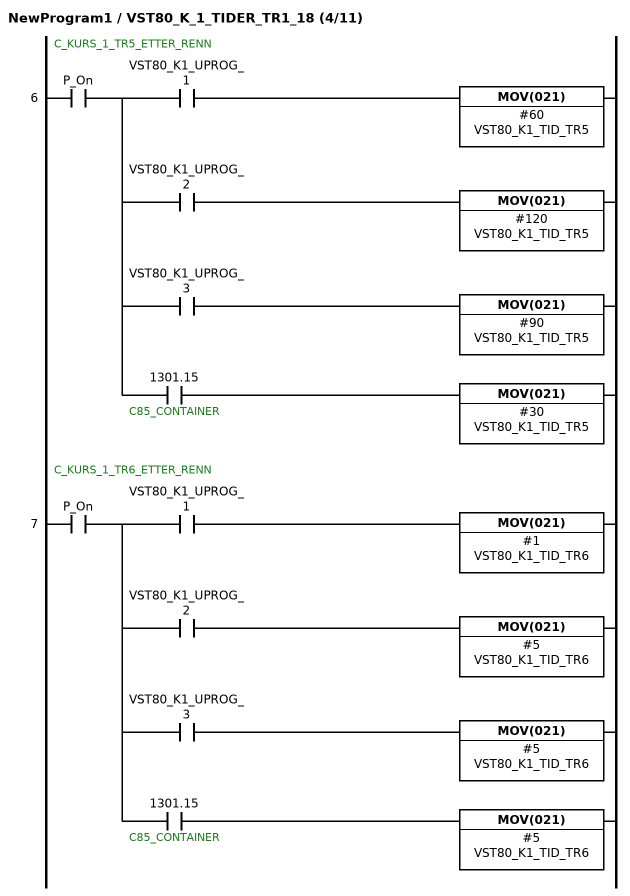
; [picture p72: NewProgram1 / VST80_K_1_TIDER_TR1_18, rungs 6-7]
; rung 6: C_KURS_1_TR5_ETTER_RENN
LD P_On
OUT TR0
AND VST80_K1_UPROG_1
MOV(021) #60 VST80_K1_TID_TR5
LD TR0
AND VST80_K1_UPROG_2
MOV(021) #120 VST80_K1_TID_TR5
LD TR0
AND VST80_K1_UPROG_3
MOV(021) #90 VST80_K1_TID_TR5
LD TR0
AND 1301.15  ; C85_CONTAINER
MOV(021) #30 VST80_K1_TID_TR5
; rung 7: C_KURS_1_TR6_ETTER_RENN
LD P_On
OUT TR0
AND VST80_K1_UPROG_1
MOV(021) #1 VST80_K1_TID_TR6
LD TR0
AND VST80_K1_UPROG_2
MOV(021) #5 VST80_K1_TID_TR6
LD TR0
AND VST80_K1_UPROG_3
MOV(021) #5 VST80_K1_TID_TR6
LD TR0
AND 1301.15  ; C85_CONTAINER
MOV(021) #5 VST80_K1_TID_TR6

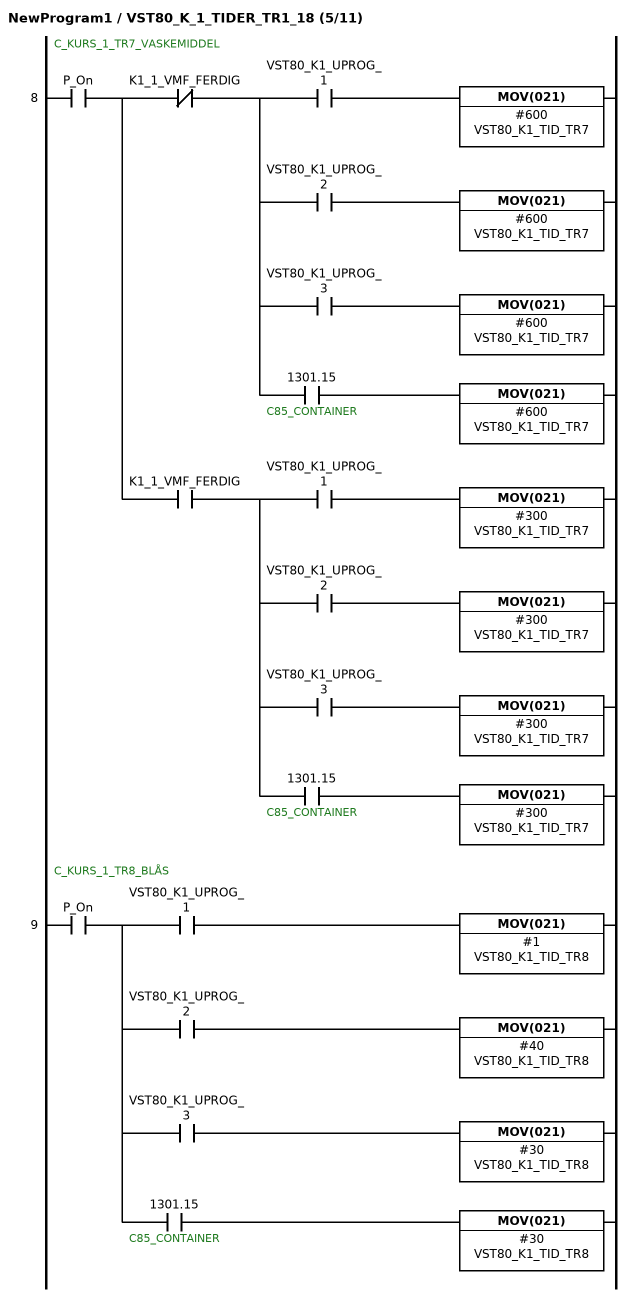
; rung 8: C_KURS_1_TR7_VASKEMIDDEL
LD P_On
OUT TR0
ANDNOT K1_1_VMF_FERDIG
OUT TR1
AND VST80_K1_UPROG_1
MOV(021) #600 VST80_K1_TID_TR7
LD TR1
AND VST80_K1_UPROG_2
MOV(021) #600 VST80_K1_TID_TR7
LD TR1
AND VST80_K1_UPROG_3
MOV(021) #600 VST80_K1_TID_TR7
LD TR1
AND 1301.15  ; C85_CONTAINER
MOV(021) #600 VST80_K1_TID_TR7
LD TR0
AND K1_1_VMF_FERDIG
OUT TR0
AND VST80_K1_UPROG_1
MOV(021) #300 VST80_K1_TID_TR7
LD TR0
AND VST80_K1_UPROG_2
MOV(021) #300 VST80_K1_TID_TR7
LD TR0
AND VST80_K1_UPROG_3
MOV(021) #300 VST80_K1_TID_TR7
LD TR0
AND 1301.15  ; C85_CONTAINER
MOV(021) #300 VST80_K1_TID_TR7
; rung 9: C_KURS_1_TR8_BLÅS
LD P_On
OUT TR0
AND VST80_K1_UPROG_1
MOV(021) #1 VST80_K1_TID_TR8
LD TR0
AND VST80_K1_UPROG_2
MOV(021) #40 VST80_K1_TID_TR8
LD TR0
AND VST80_K1_UPROG_3
MOV(021) #30 VST80_K1_TID_TR8
LD TR0
AND 1301.15  ; C85_CONTAINER
MOV(021) #30 VST80_K1_TID_TR8

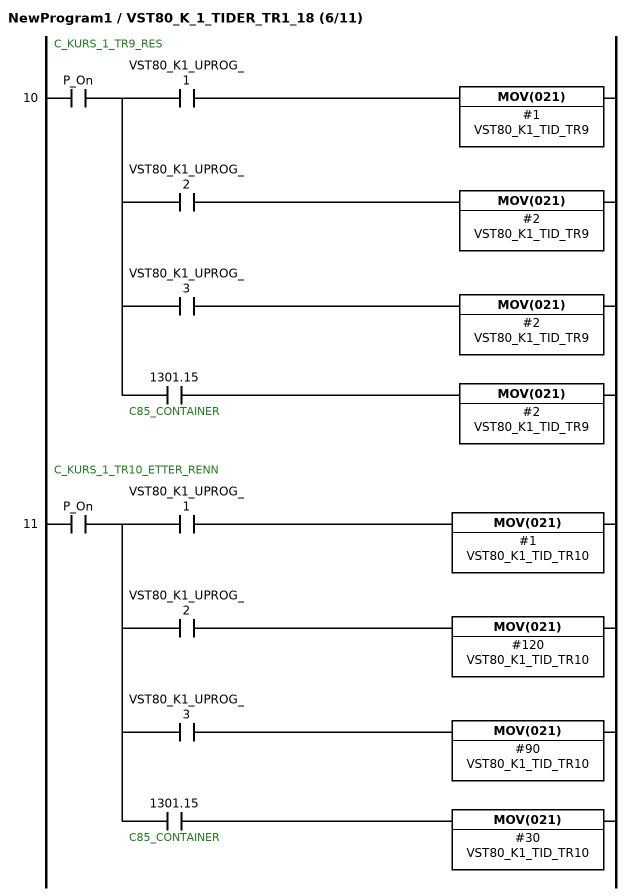
; rung 10: C_KURS_1_TR9_RES
LD P_On
OUT TR0
AND VST80_K1_UPROG_1
MOV(021) #1 VST80_K1_TID_TR9
LD TR0
AND VST80_K1_UPROG_2
MOV(021) #2 VST80_K1_TID_TR9
LD TR0
AND VST80_K1_UPROG_3
MOV(021) #2 VST80_K1_TID_TR9
LD TR0
AND 1301.15  ; C85_CONTAINER
MOV(021) #2 VST80_K1_TID_TR9
; rung 11: C_KURS_1_TR10_ETTER_RENN
LD P_On
OUT TR0
AND VST80_K1_UPROG_1
MOV(021) #1 VST80_K1_TID_TR10
LD TR0
AND VST80_K1_UPROG_2
MOV(021) #120 VST80_K1_TID_TR10
LD TR0
AND VST80_K1_UPROG_3
MOV(021) #90 VST80_K1_TID_TR10
LD TR0
AND 1301.15  ; C85_CONTAINER
MOV(021) #30 VST80_K1_TID_TR10

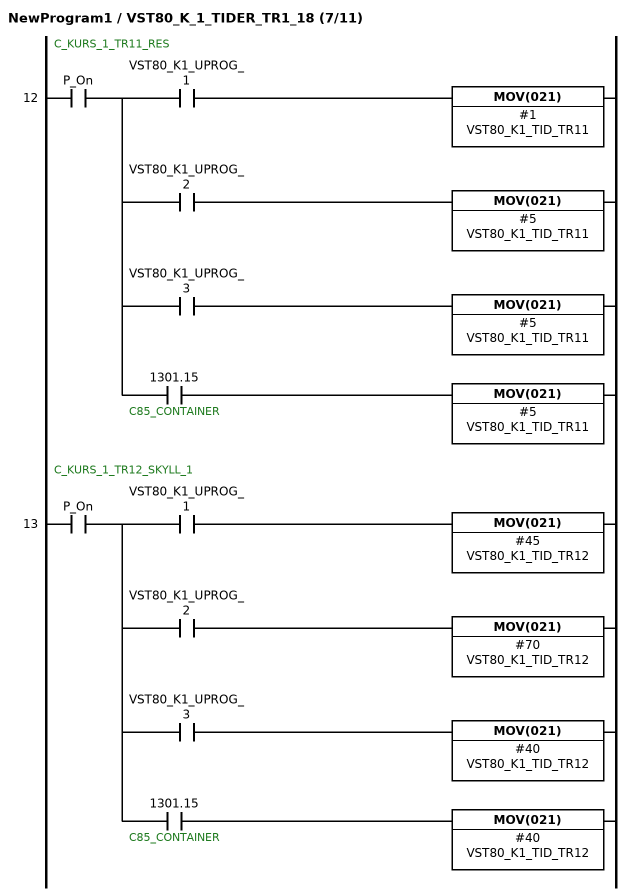
; rung 12: C_KURS_1_TR11_RES
LD P_On
OUT TR0
AND VST80_K1_UPROG_1
MOV(021) #1 VST80_K1_TID_TR11
LD TR0
AND VST80_K1_UPROG_2
MOV(021) #5 VST80_K1_TID_TR11
LD TR0
AND VST80_K1_UPROG_3
MOV(021) #5 VST80_K1_TID_TR11
LD TR0
AND 1301.15  ; C85_CONTAINER
MOV(021) #5 VST80_K1_TID_TR11
; rung 13: C_KURS_1_TR12_SKYLL_1
LD P_On
OUT TR0
AND VST80_K1_UPROG_1
MOV(021) #45 VST80_K1_TID_TR12
LD TR0
AND VST80_K1_UPROG_2
MOV(021) #70 VST80_K1_TID_TR12
LD TR0
AND VST80_K1_UPROG_3
MOV(021) #40 VST80_K1_TID_TR12
LD TR0
AND 1301.15  ; C85_CONTAINER
MOV(021) #40 VST80_K1_TID_TR12

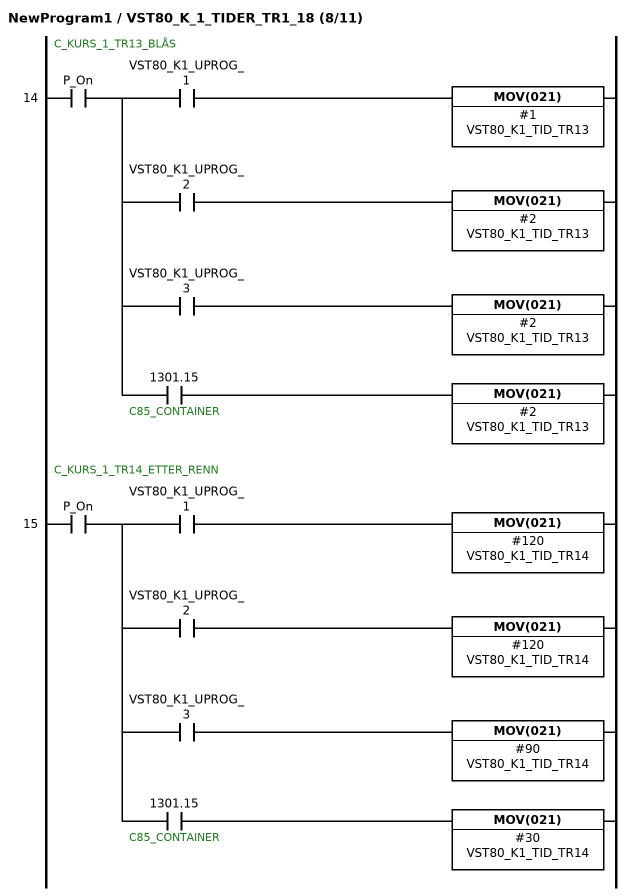
; rung 14: C_KURS_1_TR13_BLÅS
LD P_On
OUT TR0
AND VST80_K1_UPROG_1
MOV(021) #1 VST80_K1_TID_TR13
LD TR0
AND VST80_K1_UPROG_2
MOV(021) #2 VST80_K1_TID_TR13
LD TR0
AND VST80_K1_UPROG_3
MOV(021) #2 VST80_K1_TID_TR13
LD TR0
AND 1301.15  ; C85_CONTAINER
MOV(021) #2 VST80_K1_TID_TR13
; rung 15: C_KURS_1_TR14_ETTER_RENN
LD P_On
OUT TR0
AND VST80_K1_UPROG_1
MOV(021) #120 VST80_K1_TID_TR14
LD TR0
AND VST80_K1_UPROG_2
MOV(021) #120 VST80_K1_TID_TR14
LD TR0
AND VST80_K1_UPROG_3
MOV(021) #90 VST80_K1_TID_TR14
LD TR0
AND 1301.15  ; C85_CONTAINER
MOV(021) #30 VST80_K1_TID_TR14

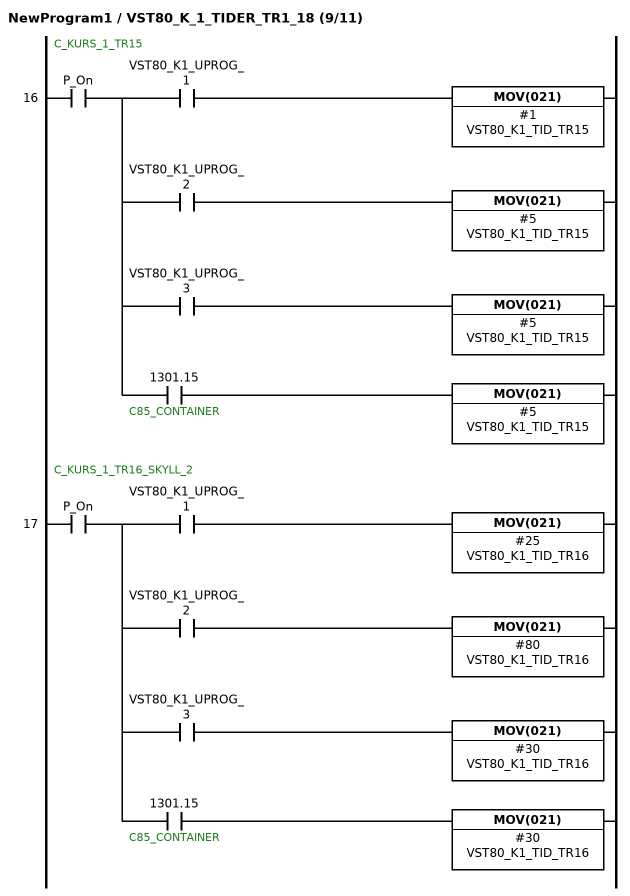
; rung 16: C_KURS_1_TR15
LD P_On
OUT TR0
AND VST80_K1_UPROG_1
MOV(021) #1 VST80_K1_TID_TR15
LD TR0
AND VST80_K1_UPROG_2
MOV(021) #5 VST80_K1_TID_TR15
LD TR0
AND VST80_K1_UPROG_3
MOV(021) #5 VST80_K1_TID_TR15
LD TR0
AND 1301.15  ; C85_CONTAINER
MOV(021) #5 VST80_K1_TID_TR15
; rung 17: C_KURS_1_TR16_SKYLL_2
LD P_On
OUT TR0
AND VST80_K1_UPROG_1
MOV(021) #25 VST80_K1_TID_TR16
LD TR0
AND VST80_K1_UPROG_2
MOV(021) #80 VST80_K1_TID_TR16
LD TR0
AND VST80_K1_UPROG_3
MOV(021) #30 VST80_K1_TID_TR16
LD TR0
AND 1301.15  ; C85_CONTAINER
MOV(021) #30 VST80_K1_TID_TR16

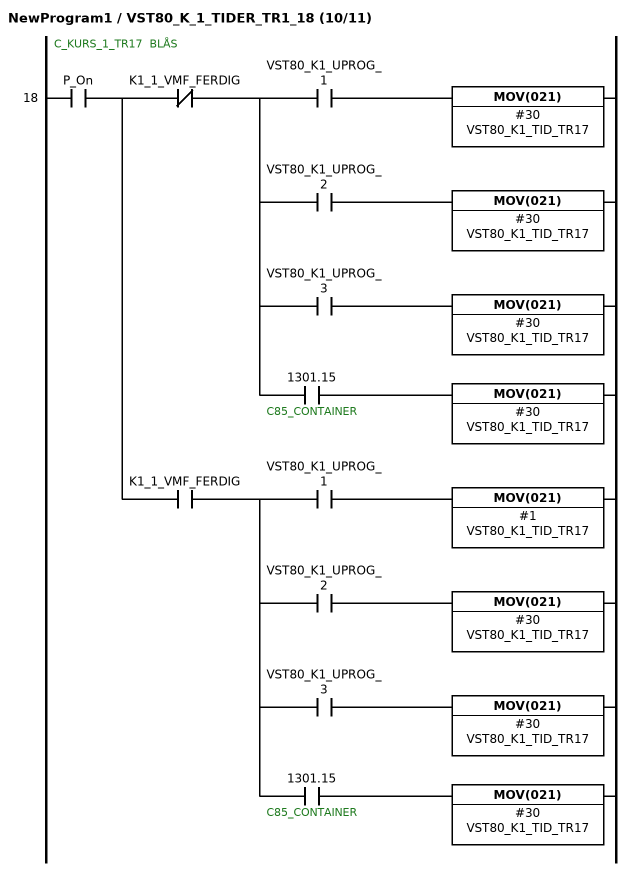
; rung 18: C_KURS_1_TR17  BLÅS
LD P_On
OUT TR0
ANDNOT K1_1_VMF_FERDIG
OUT TR1
AND VST80_K1_UPROG_1
MOV(021) #30 VST80_K1_TID_TR17
LD TR1
AND VST80_K1_UPROG_2
MOV(021) #30 VST80_K1_TID_TR17
LD TR1
AND VST80_K1_UPROG_3
MOV(021) #30 VST80_K1_TID_TR17
LD TR1
AND 1301.15  ; C85_CONTAINER
MOV(021) #30 VST80_K1_TID_TR17
LD TR0
AND K1_1_VMF_FERDIG
OUT TR0
AND VST80_K1_UPROG_1
MOV(021) #1 VST80_K1_TID_TR17
LD TR0
AND VST80_K1_UPROG_2
MOV(021) #30 VST80_K1_TID_TR17
LD TR0
AND VST80_K1_UPROG_3
MOV(021) #30 VST80_K1_TID_TR17
LD TR0
AND 1301.15  ; C85_CONTAINER
MOV(021) #30 VST80_K1_TID_TR17

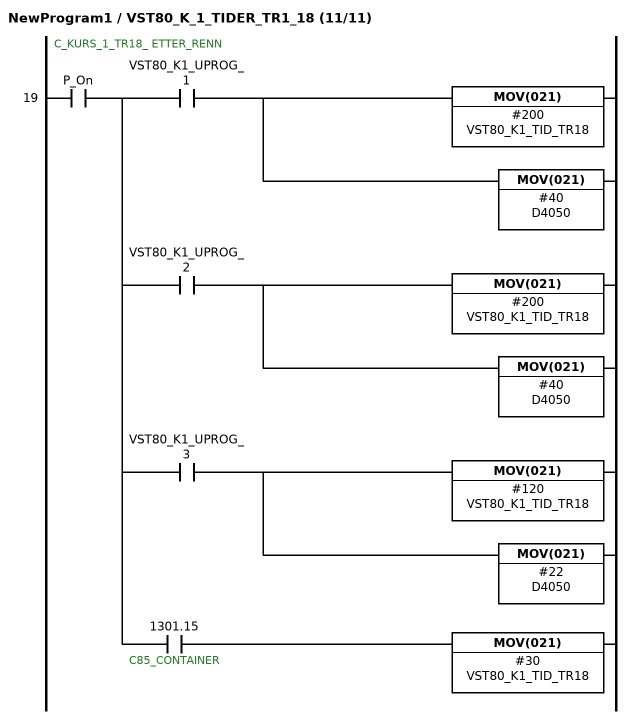
; rung 19: C_KURS_1_TR18_ ETTER_RENN
LD P_On
OUT TR0
AND VST80_K1_UPROG_1
MOV(021) #200 VST80_K1_TID_TR18
MOV(021) #40 D4050
LD TR0
AND VST80_K1_UPROG_2
MOV(021) #200 VST80_K1_TID_TR18
MOV(021) #40 D4050
LD TR0
AND VST80_K1_UPROG_3
MOV(021) #120 VST80_K1_TID_TR18
MOV(021) #22 D4050
LD TR0
AND 1301.15  ; C85_CONTAINER
MOV(021) #30 VST80_K1_TID_TR18

### Section VST80_K_1_TIDER_TR19_30

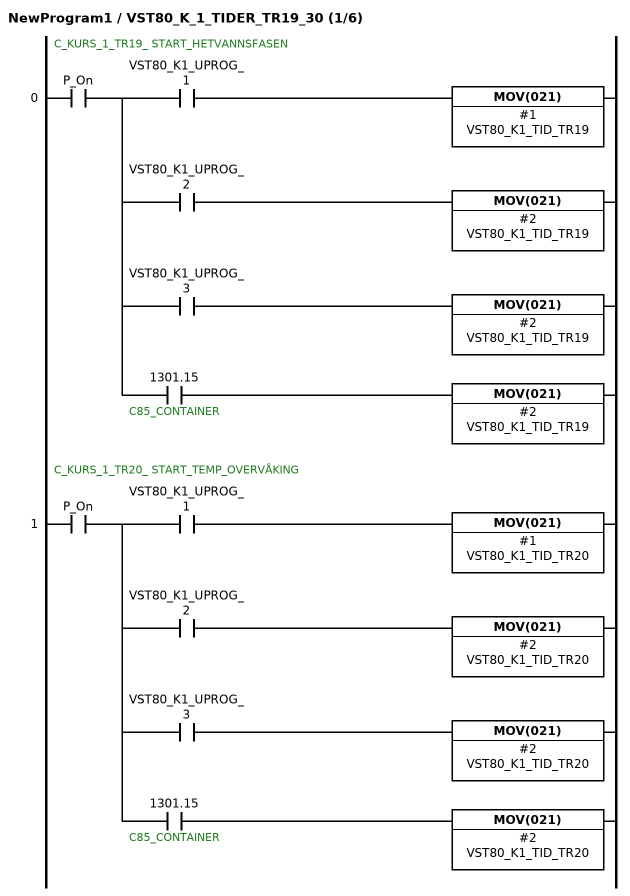
; rung 0: C_KURS_1_TR19_ START_HETVANNSFASEN
LD P_On
OUT TR0
AND VST80_K1_UPROG_1
MOV(021) #1 VST80_K1_TID_TR19
LD TR0
AND VST80_K1_UPROG_2
MOV(021) #2 VST80_K1_TID_TR19
LD TR0
AND VST80_K1_UPROG_3
MOV(021) #2 VST80_K1_TID_TR19
LD TR0
AND 1301.15  ; C85_CONTAINER
MOV(021) #2 VST80_K1_TID_TR19
; rung 1: C_KURS_1_TR20_ START_TEMP_OVERVÅKING
LD P_On
OUT TR0
AND VST80_K1_UPROG_1
MOV(021) #1 VST80_K1_TID_TR20
LD TR0
AND VST80_K1_UPROG_2
MOV(021) #2 VST80_K1_TID_TR20
LD TR0
AND VST80_K1_UPROG_3
MOV(021) #2 VST80_K1_TID_TR20
LD TR0
AND 1301.15  ; C85_CONTAINER
MOV(021) #2 VST80_K1_TID_TR20

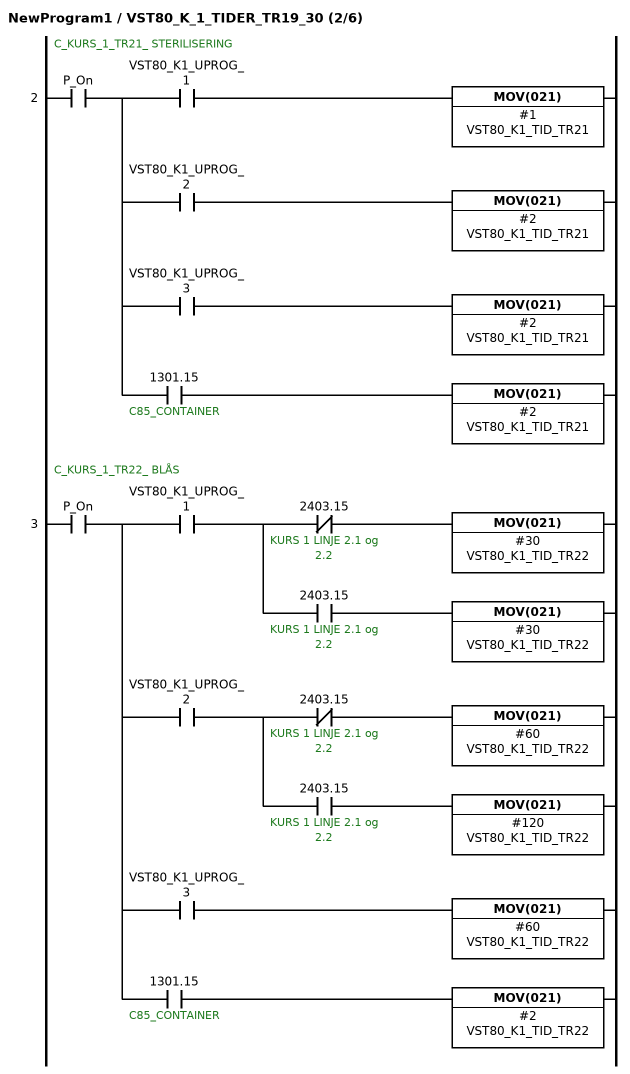
; rung 2: C_KURS_1_TR21_ STERILISERING
LD P_On
OUT TR0
AND VST80_K1_UPROG_1
MOV(021) #1 VST80_K1_TID_TR21
LD TR0
AND VST80_K1_UPROG_2
MOV(021) #2 VST80_K1_TID_TR21
LD TR0
AND VST80_K1_UPROG_3
MOV(021) #2 VST80_K1_TID_TR21
LD TR0
AND 1301.15  ; C85_CONTAINER
MOV(021) #2 VST80_K1_TID_TR21
; rung 3: C_KURS_1_TR22_ BLÅS
LD P_On
OUT TR0
AND VST80_K1_UPROG_1
OUT TR1
ANDNOT 2403.15  ; KURS 1 LINJE 2.1 og 2.2
MOV(021) #30 VST80_K1_TID_TR22
LD TR1
AND 2403.15  ; KURS 1 LINJE 2.1 og 2.2
MOV(021) #30 VST80_K1_TID_TR22
LD TR0
AND VST80_K1_UPROG_2
OUT TR1
ANDNOT 2403.15  ; KURS 1 LINJE 2.1 og 2.2
MOV(021) #60 VST80_K1_TID_TR22
LD TR1
AND 2403.15  ; KURS 1 LINJE 2.1 og 2.2
MOV(021) #120 VST80_K1_TID_TR22
LD TR0
AND VST80_K1_UPROG_3
MOV(021) #60 VST80_K1_TID_TR22
LD TR0
AND 1301.15  ; C85_CONTAINER
MOV(021) #2 VST80_K1_TID_TR22

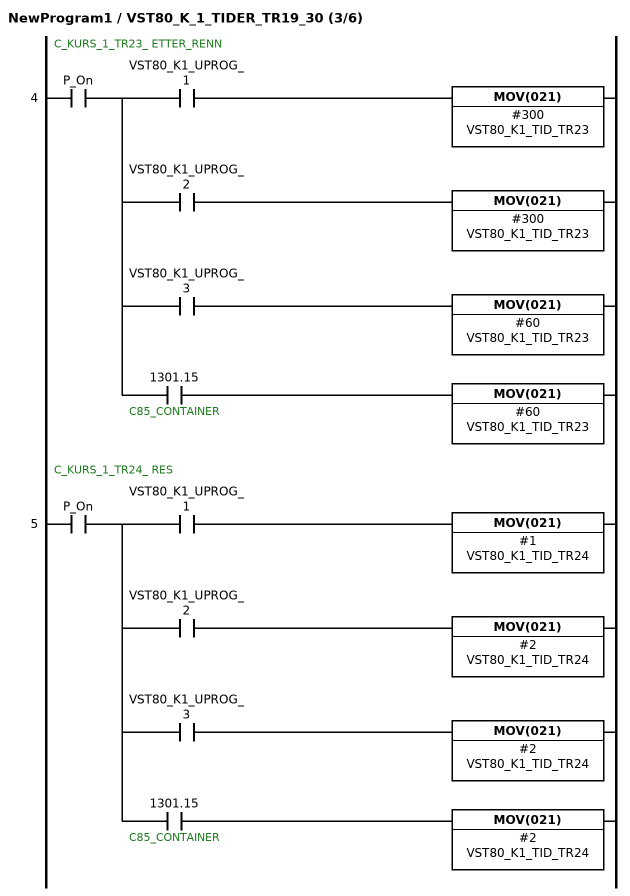
; rung 4: C_KURS_1_TR23_ ETTER_RENN
LD P_On
OUT TR0
AND VST80_K1_UPROG_1
MOV(021) #300 VST80_K1_TID_TR23
LD TR0
AND VST80_K1_UPROG_2
MOV(021) #300 VST80_K1_TID_TR23
LD TR0
AND VST80_K1_UPROG_3
MOV(021) #60 VST80_K1_TID_TR23
LD TR0
AND 1301.15  ; C85_CONTAINER
MOV(021) #60 VST80_K1_TID_TR23
; rung 5: C_KURS_1_TR24_ RES
LD P_On
OUT TR0
AND VST80_K1_UPROG_1
MOV(021) #1 VST80_K1_TID_TR24
LD TR0
AND VST80_K1_UPROG_2
MOV(021) #2 VST80_K1_TID_TR24
LD TR0
AND VST80_K1_UPROG_3
MOV(021) #2 VST80_K1_TID_TR24
LD TR0
AND 1301.15  ; C85_CONTAINER
MOV(021) #2 VST80_K1_TID_TR24

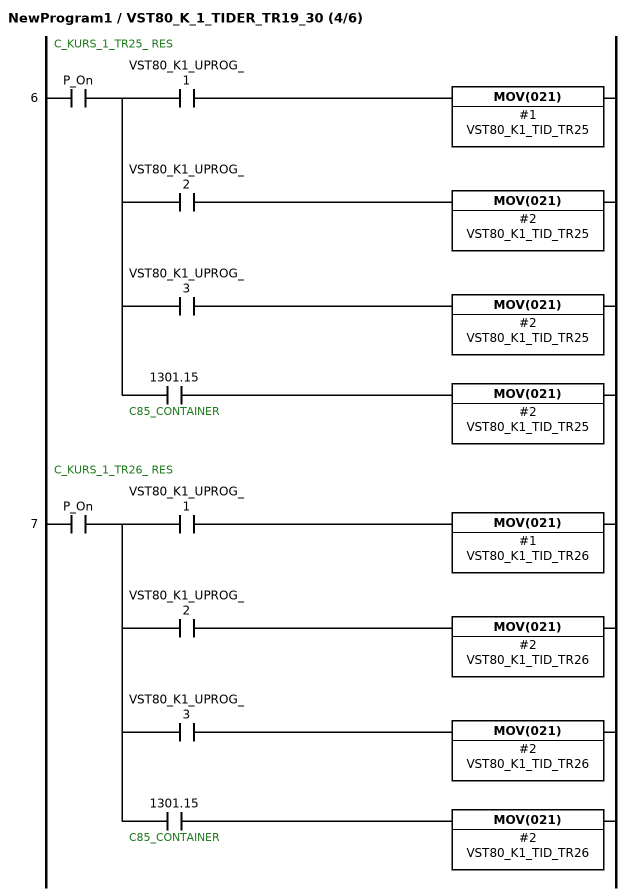
; rung 6: C_KURS_1_TR25_ RES
LD P_On
OUT TR0
AND VST80_K1_UPROG_1
MOV(021) #1 VST80_K1_TID_TR25
LD TR0
AND VST80_K1_UPROG_2
MOV(021) #2 VST80_K1_TID_TR25
LD TR0
AND VST80_K1_UPROG_3
MOV(021) #2 VST80_K1_TID_TR25
LD TR0
AND 1301.15  ; C85_CONTAINER
MOV(021) #2 VST80_K1_TID_TR25
; rung 7: C_KURS_1_TR26_ RES
LD P_On
OUT TR0
AND VST80_K1_UPROG_1
MOV(021) #1 VST80_K1_TID_TR26
LD TR0
AND VST80_K1_UPROG_2
MOV(021) #2 VST80_K1_TID_TR26
LD TR0
AND VST80_K1_UPROG_3
MOV(021) #2 VST80_K1_TID_TR26
LD TR0
AND 1301.15  ; C85_CONTAINER
MOV(021) #2 VST80_K1_TID_TR26

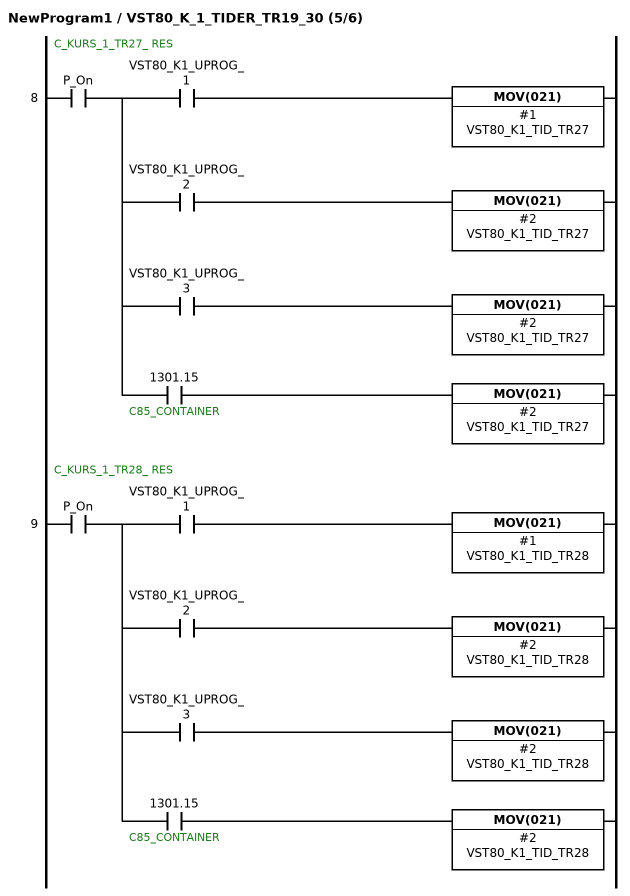
; rung 8: C_KURS_1_TR27_ RES
LD P_On
OUT TR0
AND VST80_K1_UPROG_1
MOV(021) #1 VST80_K1_TID_TR27
LD TR0
AND VST80_K1_UPROG_2
MOV(021) #2 VST80_K1_TID_TR27
LD TR0
AND VST80_K1_UPROG_3
MOV(021) #2 VST80_K1_TID_TR27
LD TR0
AND 1301.15  ; C85_CONTAINER
MOV(021) #2 VST80_K1_TID_TR27
; rung 9: C_KURS_1_TR28_ RES
LD P_On
OUT TR0
AND VST80_K1_UPROG_1
MOV(021) #1 VST80_K1_TID_TR28
LD TR0
AND VST80_K1_UPROG_2
MOV(021) #2 VST80_K1_TID_TR28
LD TR0
AND VST80_K1_UPROG_3
MOV(021) #2 VST80_K1_TID_TR28
LD TR0
AND 1301.15  ; C85_CONTAINER
MOV(021) #2 VST80_K1_TID_TR28

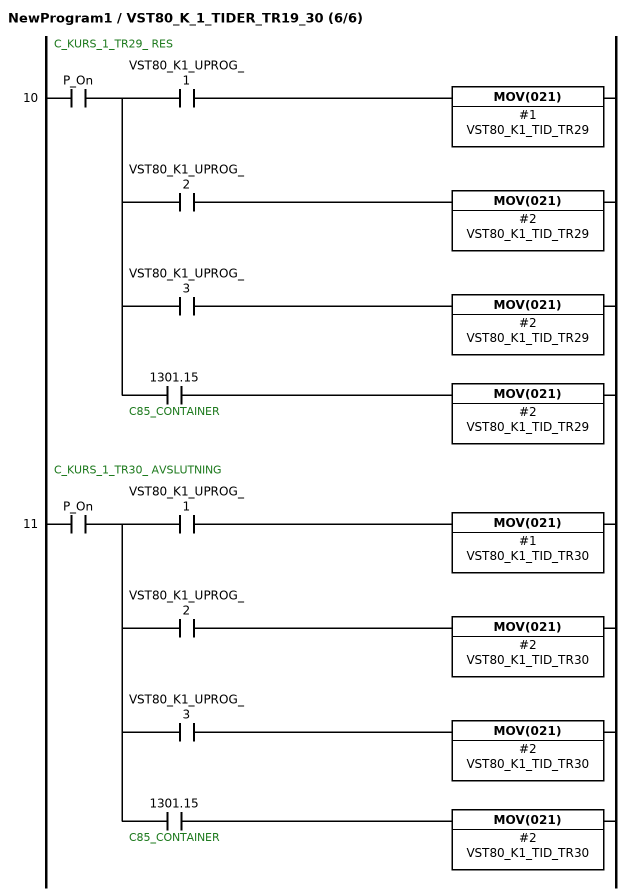
; rung 10: C_KURS_1_TR29_ RES
LD P_On
OUT TR0
AND VST80_K1_UPROG_1
MOV(021) #1 VST80_K1_TID_TR29
LD TR0
AND VST80_K1_UPROG_2
MOV(021) #2 VST80_K1_TID_TR29
LD TR0
AND VST80_K1_UPROG_3
MOV(021) #2 VST80_K1_TID_TR29
LD TR0
AND 1301.15  ; C85_CONTAINER
MOV(021) #2 VST80_K1_TID_TR29
; rung 11: C_KURS_1_TR30_ AVSLUTNING
LD P_On
OUT TR0
AND VST80_K1_UPROG_1
MOV(021) #1 VST80_K1_TID_TR30
LD TR0
AND VST80_K1_UPROG_2
MOV(021) #2 VST80_K1_TID_TR30
LD TR0
AND VST80_K1_UPROG_3
MOV(021) #2 VST80_K1_TID_TR30
LD TR0
AND 1301.15  ; C85_CONTAINER
MOV(021) #2 VST80_K1_TID_TR30

### Section VST80_K1_TRINN
; Vaskeprogrammet består av 30. hovedtrinn. / Funksjonsbenstabell: 975100-BL48

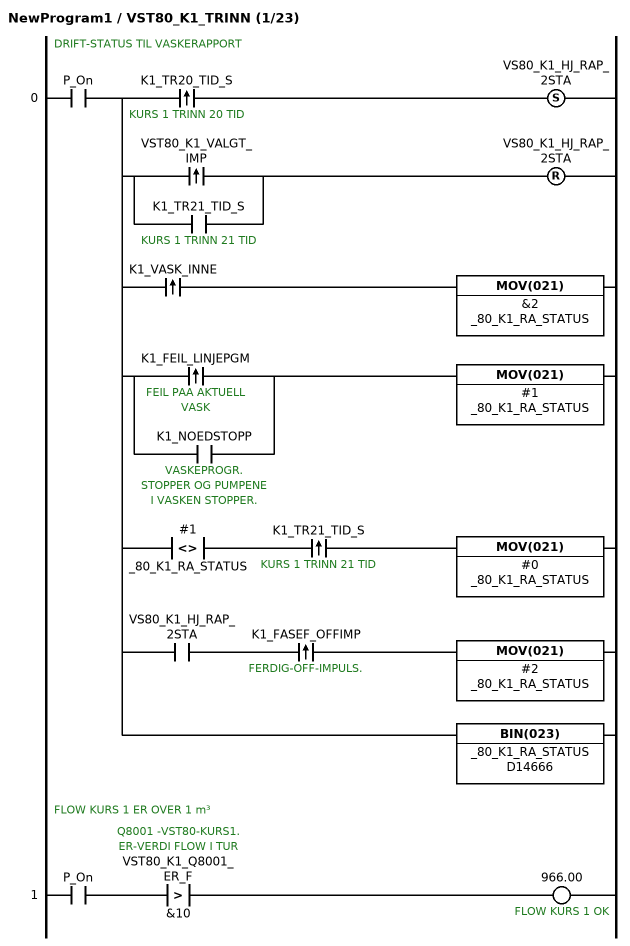
; rung 0: DRIFT-STATUS TIL VASKERAPPORT
LD P_On
OUT TR0
@AND K1_TR20_TID_S  ; KURS 1 TRINN 20 TID
SET VS80_K1_HJ_RAP_2STA
LD TR0
@LD VST80_K1_VALGT_IMP
OR K1_TR21_TID_S  ; KURS 1 TRINN 21 TID
ANDLD
RSET VS80_K1_HJ_RAP_2STA
LD TR0
@AND K1_VASK_INNE
MOV(021) &2 _80_K1_RA_STATUS
LD TR0
@LD K1_FEIL_LINJEPGM  ; FEIL PAA AKTUELL VASK
OR K1_NOEDSTOPP  ; VASKEPROGR. STOPPER OG PUMPENE I VASKEN STOPPER.
ANDLD
MOV(021) #1 _80_K1_RA_STATUS
LD TR0
AND<>(305) #1 _80_K1_RA_STATUS
@AND K1_TR21_TID_S  ; KURS 1 TRINN 21 TID
MOV(021) #0 _80_K1_RA_STATUS
LD TR0
AND VS80_K1_HJ_RAP_2STA
@AND K1_FASEF_OFFIMP  ; FERDIG-OFF-IMPULS.
MOV(021) #2 _80_K1_RA_STATUS
LD TR0
BIN(023) _80_K1_RA_STATUS D14666
; rung 1: FLOW KURS 1 ER OVER 1 m³
LD P_On
AND>(320) VST80_K1_Q8001_ER_F &10  ; Q8001 -VST80-KURS1. ER-VERDI FLOW I TUR
OUT 966.00  ; FLOW KURS 1 OK

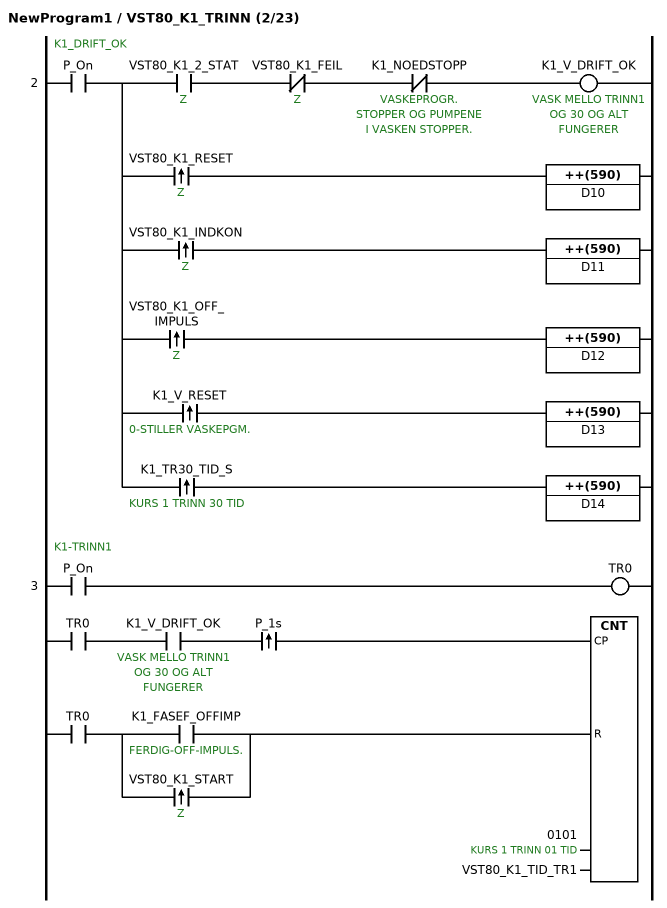
; rung 2: K1_DRIFT_OK
LD P_On
OUT TR0
AND VST80_K1_2_STAT  ; Z
ANDNOT VST80_K1_FEIL  ; Z
ANDNOT K1_NOEDSTOPP  ; VASKEPROGR. STOPPER OG PUMPENE I VASKEN STOPPER.
OUT K1_V_DRIFT_OK  ; VASK MELLO TRINN1 OG 30 OG ALT FUNGERER
LD TR0
@AND VST80_K1_RESET  ; Z
++(590) D10
LD TR0
@AND VST80_K1_INDKON  ; Z
++(590) D11
LD TR0
@AND VST80_K1_OFF_IMPULS  ; Z
++(590) D12
LD TR0
@AND K1_V_RESET  ; 0-STILLER VASKEPGM.
++(590) D13
LD TR0
@AND K1_TR30_TID_S  ; KURS 1 TRINN 30 TID
++(590) D14
; rung 3: K1-TRINN1
LD P_On
OUT TR0
AND K1_V_DRIFT_OK  ; VASK MELLO TRINN1 OG 30 OG ALT FUNGERER
@AND P_1s
LD TR0
LD K1_FASEF_OFFIMP  ; FERDIG-OFF-IMPULS.
@OR VST80_K1_START  ; Z
ANDLD
CNT 0101 VST80_K1_TID_TR1  ; KURS 1 TRINN 01 TID

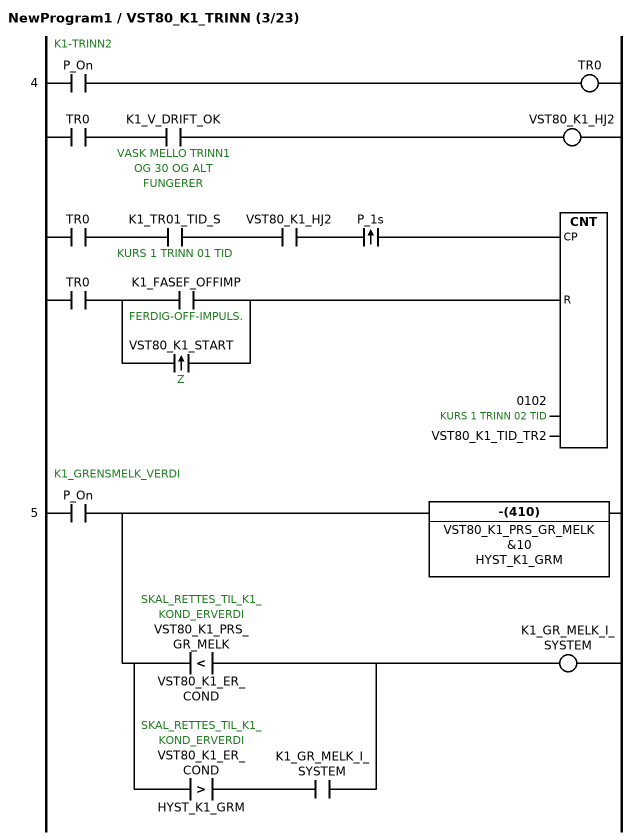
; rung 4: K1-TRINN2
LD P_On
OUT TR0
AND K1_V_DRIFT_OK  ; VASK MELLO TRINN1 OG 30 OG ALT FUNGERER
OUT VST80_K1_HJ2
LD TR0
AND K1_TR01_TID_S  ; KURS 1 TRINN 01 TID
AND VST80_K1_HJ2
@AND P_1s
LD TR0
LD K1_FASEF_OFFIMP  ; FERDIG-OFF-IMPULS.
@OR VST80_K1_START  ; Z
ANDLD
CNT 0102 VST80_K1_TID_TR2  ; KURS 1 TRINN 02 TID
; rung 5: K1_GRENSMELK_VERDI
LD P_On
-(410) VST80_K1_PRS_GR_MELK &10 HYST_K1_GRM
LD<(310) VST80_K1_PRS_GR_MELK VST80_K1_ER_COND  ; SKAL_RETTES_TIL_K1_KOND_ERVERDI
LD>(320) VST80_K1_ER_COND HYST_K1_GRM  ; SKAL_RETTES_TIL_K1_KOND_ERVERDI
AND K1_GR_MELK_I_SYSTEM
ORLD
ANDLD
OUT K1_GR_MELK_I_SYSTEM

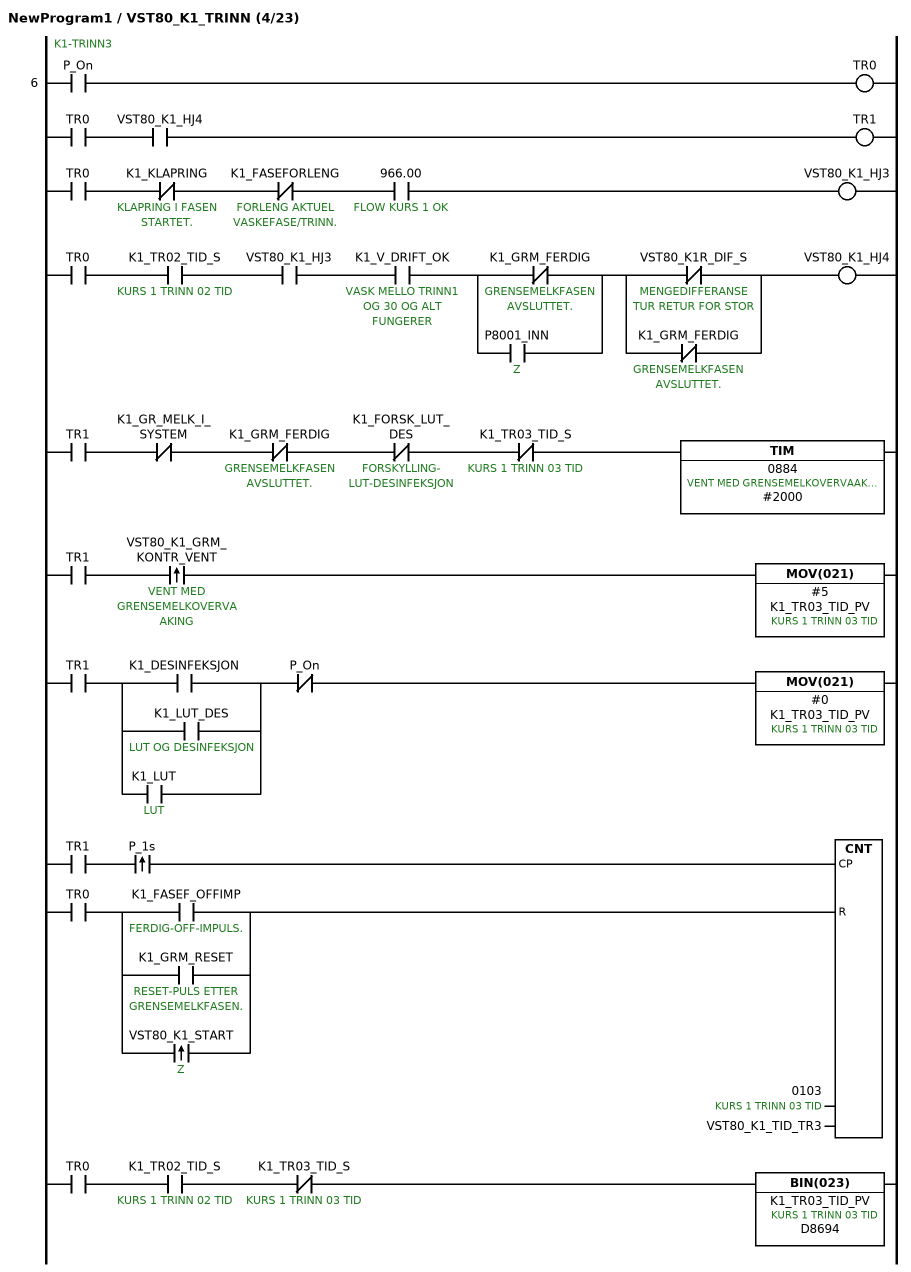
; rung 6: K1-TRINN3
LD P_On
OUT TR0
ANDNOT K1_KLAPRING  ; KLAPRING I FASEN STARTET.
ANDNOT K1_FASEFORLENG  ; FORLENG AKTUEL VASKEFASE/TRINN.
AND 966.00  ; FLOW KURS 1 OK
OUT VST80_K1_HJ3
LD TR0
AND K1_TR02_TID_S  ; KURS 1 TRINN 02 TID
AND VST80_K1_HJ3
AND K1_V_DRIFT_OK  ; VASK MELLO TRINN1 OG 30 OG ALT FUNGERER
LDNOT K1_GRM_FERDIG  ; GRENSEMELKFASEN AVSLUTTET.
OR P8001_INN  ; Z
ANDLD
LDNOT VST80_K1R_DIF_S  ; MENGEDIFFERANSE TUR RETUR FOR STOR
ORNOT K1_GRM_FERDIG  ; GRENSEMELKFASEN AVSLUTTET.
ANDLD
OUT VST80_K1_HJ4
LD TR0
AND VST80_K1_HJ4
OUT TR1
ANDNOT K1_GR_MELK_I_SYSTEM
ANDNOT K1_GRM_FERDIG  ; GRENSEMELKFASEN AVSLUTTET.
ANDNOT K1_FORSK_LUT_DES  ; FORSKYLLING- LUT-DESINFEKSJON
ANDNOT K1_TR03_TID_S  ; KURS 1 TRINN 03 TID
TIM 0884 #2000  ; VENT MED GRENSEMELKOVERVAAKING
LD TR1
@AND VST80_K1_GRM_KONTR_VENT  ; VENT MED GRENSEMELKOVERVAAKING
MOV(021) #5 K1_TR03_TID_PV  ; KURS 1 TRINN 03 TID
LD TR1
LD K1_DESINFEKSJON
OR K1_LUT_DES  ; LUT OG DESINFEKSJON
OR K1_LUT  ; LUT
ANDLD
ANDNOT P_On
MOV(021) #0 K1_TR03_TID_PV  ; KURS 1 TRINN 03 TID
LD TR1
@AND P_1s
LD TR0
LD K1_FASEF_OFFIMP  ; FERDIG-OFF-IMPULS.
OR K1_GRM_RESET  ; RESET-PULS ETTER GRENSEMELKFASEN.
@OR VST80_K1_START  ; Z
ANDLD
CNT 0103 VST80_K1_TID_TR3  ; KURS 1 TRINN 03 TID
LD TR0
AND K1_TR02_TID_S  ; KURS 1 TRINN 02 TID
ANDNOT K1_TR03_TID_S  ; KURS 1 TRINN 03 TID
BIN(023) K1_TR03_TID_PV D8694  ; KURS 1 TRINN 03 TID

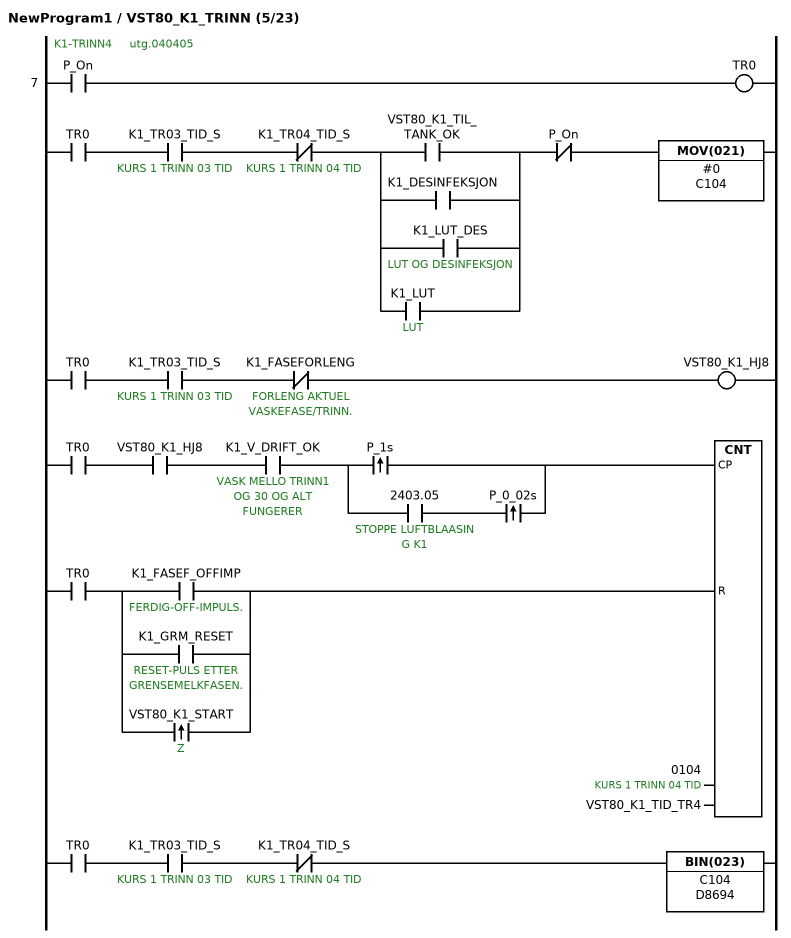
; rung 7: K1-TRINN4     utg.040405
LD P_On
OUT TR0
AND K1_TR03_TID_S  ; KURS 1 TRINN 03 TID
ANDNOT K1_TR04_TID_S  ; KURS 1 TRINN 04 TID
LD VST80_K1_TIL_TANK_OK
OR K1_DESINFEKSJON
OR K1_LUT_DES  ; LUT OG DESINFEKSJON
OR K1_LUT  ; LUT
ANDLD
ANDNOT P_On
MOV(021) #0 C104
LD TR0
AND K1_TR03_TID_S  ; KURS 1 TRINN 03 TID
ANDNOT K1_FASEFORLENG  ; FORLENG AKTUEL VASKEFASE/TRINN.
OUT VST80_K1_HJ8
LD TR0
AND VST80_K1_HJ8
AND K1_V_DRIFT_OK  ; VASK MELLO TRINN1 OG 30 OG ALT FUNGERER
@LD P_1s
LD 2403.05  ; STOPPE LUFTBLAASING K1
@AND P_0_02s
ORLD
ANDLD
LD TR0
LD K1_FASEF_OFFIMP  ; FERDIG-OFF-IMPULS.
OR K1_GRM_RESET  ; RESET-PULS ETTER GRENSEMELKFASEN.
@OR VST80_K1_START  ; Z
ANDLD
CNT 0104 VST80_K1_TID_TR4  ; KURS 1 TRINN 04 TID
LD TR0
AND K1_TR03_TID_S  ; KURS 1 TRINN 03 TID
ANDNOT K1_TR04_TID_S  ; KURS 1 TRINN 04 TID
BIN(023) C104 D8694

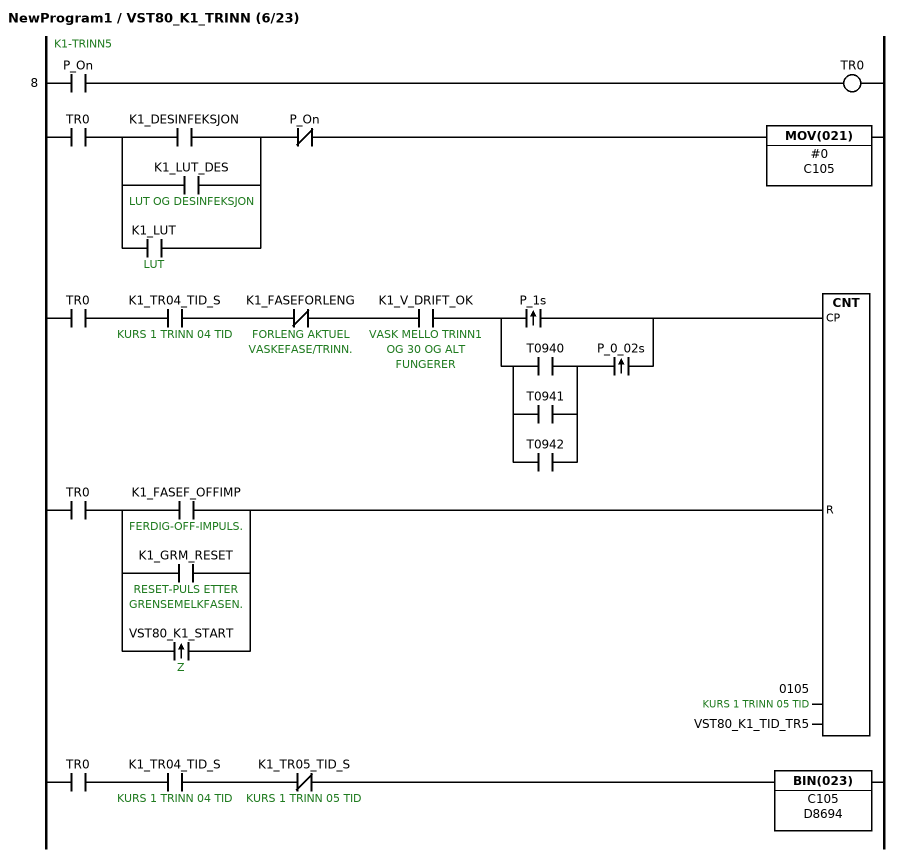
; rung 8: K1-TRINN5
LD P_On
OUT TR0
LD K1_DESINFEKSJON
OR K1_LUT_DES  ; LUT OG DESINFEKSJON
OR K1_LUT  ; LUT
ANDLD
ANDNOT P_On
MOV(021) #0 C105
LD TR0
AND K1_TR04_TID_S  ; KURS 1 TRINN 04 TID
ANDNOT K1_FASEFORLENG  ; FORLENG AKTUEL VASKEFASE/TRINN.
AND K1_V_DRIFT_OK  ; VASK MELLO TRINN1 OG 30 OG ALT FUNGERER
@LD P_1s
LD T0940
OR T0941
OR T0942
@AND P_0_02s
ORLD
ANDLD
LD TR0
LD K1_FASEF_OFFIMP  ; FERDIG-OFF-IMPULS.
OR K1_GRM_RESET  ; RESET-PULS ETTER GRENSEMELKFASEN.
@OR VST80_K1_START  ; Z
ANDLD
CNT 0105 VST80_K1_TID_TR5  ; KURS 1 TRINN 05 TID
LD TR0
AND K1_TR04_TID_S  ; KURS 1 TRINN 04 TID
ANDNOT K1_TR05_TID_S  ; KURS 1 TRINN 05 TID
BIN(023) C105 D8694

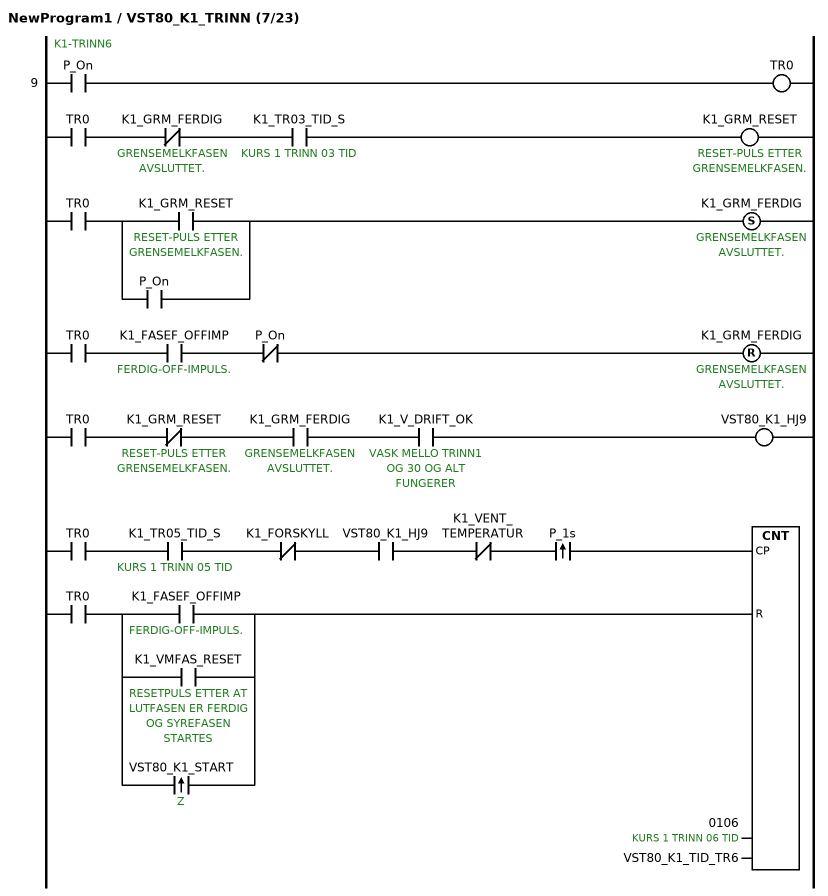
; rung 9: K1-TRINN6
LD P_On
OUT TR0
ANDNOT K1_GRM_FERDIG  ; GRENSEMELKFASEN AVSLUTTET.
AND K1_TR03_TID_S  ; KURS 1 TRINN 03 TID
OUT K1_GRM_RESET  ; RESET-PULS ETTER GRENSEMELKFASEN.
LD TR0
LD K1_GRM_RESET  ; RESET-PULS ETTER GRENSEMELKFASEN.
OR P_On
ANDLD
SET K1_GRM_FERDIG  ; GRENSEMELKFASEN AVSLUTTET.
LD TR0
AND K1_FASEF_OFFIMP  ; FERDIG-OFF-IMPULS.
ANDNOT P_On
RSET K1_GRM_FERDIG  ; GRENSEMELKFASEN AVSLUTTET.
LD TR0
ANDNOT K1_GRM_RESET  ; RESET-PULS ETTER GRENSEMELKFASEN.
AND K1_GRM_FERDIG  ; GRENSEMELKFASEN AVSLUTTET.
AND K1_V_DRIFT_OK  ; VASK MELLO TRINN1 OG 30 OG ALT FUNGERER
OUT VST80_K1_HJ9
LD TR0
AND K1_TR05_TID_S  ; KURS 1 TRINN 05 TID
ANDNOT K1_FORSKYLL
AND VST80_K1_HJ9
ANDNOT K1_VENT_TEMPERATUR
@AND P_1s
LD TR0
LD K1_FASEF_OFFIMP  ; FERDIG-OFF-IMPULS.
OR K1_VMFAS_RESET  ; RESETPULS ETTER AT LUTFASEN ER FERDIG OG SYREFASEN STARTES
@OR VST80_K1_START  ; Z
ANDLD
CNT 0106 VST80_K1_TID_TR6  ; KURS 1 TRINN 06 TID

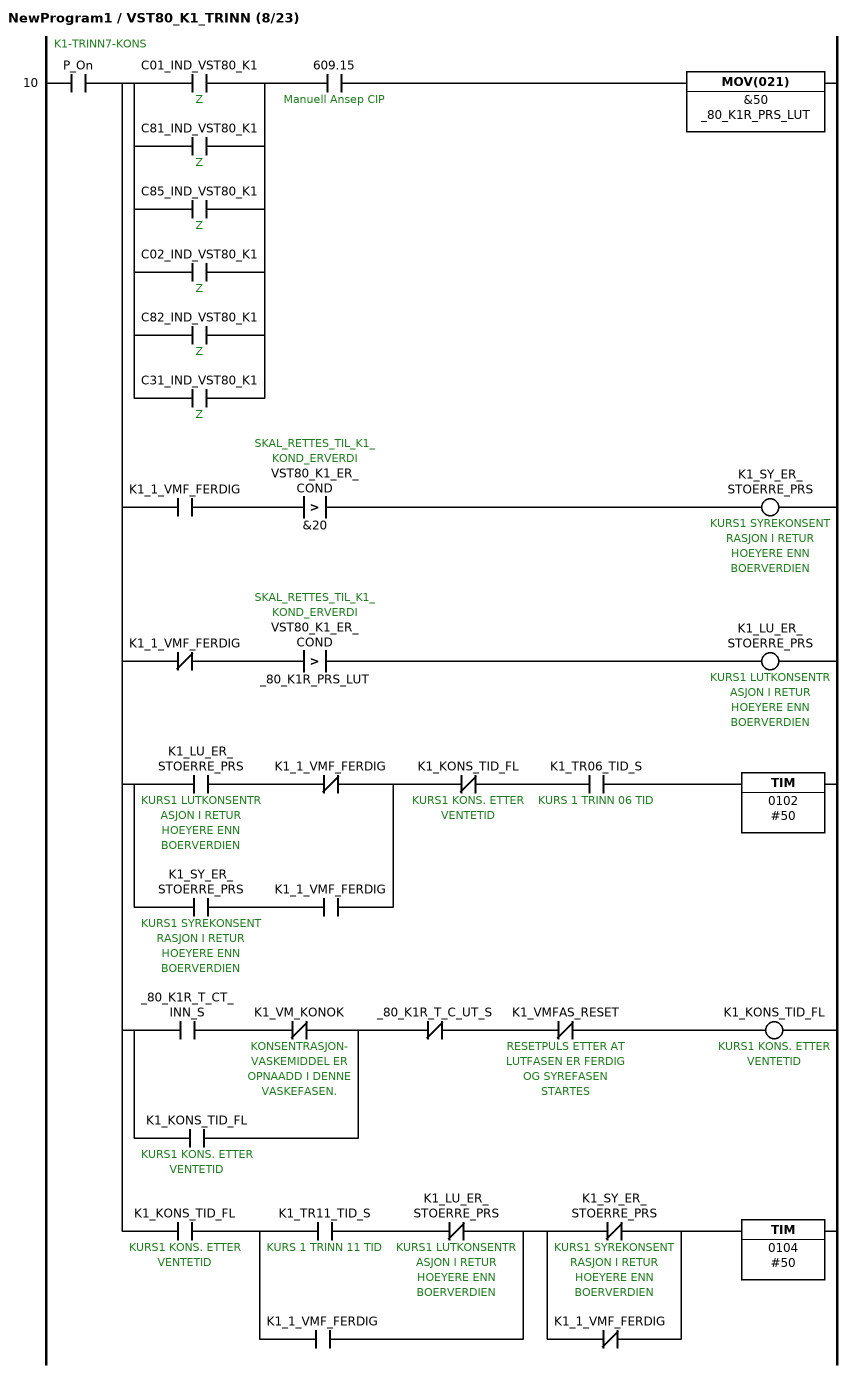
; rung 10: K1-TRINN7-KONS
LD P_On
OUT TR0
LD C01_IND_VST80_K1  ; Z
OR C81_IND_VST80_K1  ; Z
OR C85_IND_VST80_K1  ; Z
OR C02_IND_VST80_K1  ; Z
OR C82_IND_VST80_K1  ; Z
OR C31_IND_VST80_K1  ; Z
ANDLD
AND 609.15  ; Manuell Ansep CIP
MOV(021) &50 _80_K1R_PRS_LUT
LD TR0
AND K1_1_VMF_FERDIG
AND>(320) VST80_K1_ER_COND &20  ; SKAL_RETTES_TIL_K1_KOND_ERVERDI
OUT K1_SY_ER_STOERRE_PRS  ; KURS1 SYREKONSENTRASJON I RETUR HOEYERE ENN BOERVERDIEN
LD TR0
ANDNOT K1_1_VMF_FERDIG
AND>(320) VST80_K1_ER_COND _80_K1R_PRS_LUT  ; SKAL_RETTES_TIL_K1_KOND_ERVERDI
OUT K1_LU_ER_STOERRE_PRS  ; KURS1 LUTKONSENTRASJON I RETUR HOEYERE ENN BOERVERDIEN
LD TR0
LD K1_LU_ER_STOERRE_PRS  ; KURS1 LUTKONSENTRASJON I RETUR HOEYERE ENN BOERVERDIEN
ANDNOT K1_1_VMF_FERDIG
LD K1_SY_ER_STOERRE_PRS  ; KURS1 SYREKONSENTRASJON I RETUR HOEYERE ENN BOERVERDIEN
AND K1_1_VMF_FERDIG
ORLD
ANDLD
ANDNOT K1_KONS_TID_FL  ; KURS1 KONS. ETTER VENTETID
AND K1_TR06_TID_S  ; KURS 1 TRINN 06 TID
TIM 0102 #50
LD TR0
LD _80_K1R_T_CT_INN_S
ANDNOT K1_VM_KONOK  ; KONSENTRASJON-VASKEMIDDEL ER OPNAADD I DENNE VASKEFASEN.
OR K1_KONS_TID_FL  ; KURS1 KONS. ETTER VENTETID
ANDLD
ANDNOT _80_K1R_T_C_UT_S
ANDNOT K1_VMFAS_RESET  ; RESETPULS ETTER AT LUTFASEN ER FERDIG OG SYREFASEN STARTES
OUT K1_KONS_TID_FL  ; KURS1 KONS. ETTER VENTETID
LD TR0
AND K1_KONS_TID_FL  ; KURS1 KONS. ETTER VENTETID
LD K1_TR11_TID_S  ; KURS 1 TRINN 11 TID
ANDNOT K1_LU_ER_STOERRE_PRS  ; KURS1 LUTKONSENTRASJON I RETUR HOEYERE ENN BOERVERDIEN
OR K1_1_VMF_FERDIG
ANDLD
LDNOT K1_SY_ER_STOERRE_PRS  ; KURS1 SYREKONSENTRASJON I RETUR HOEYERE ENN BOERVERDIEN
ORNOT K1_1_VMF_FERDIG
ANDLD
TIM 0104 #50

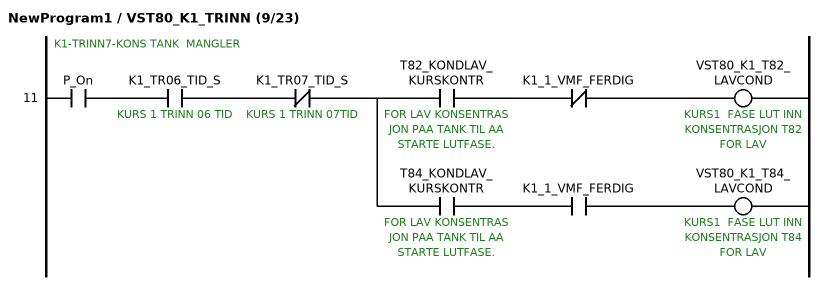
; rung 11: K1-TRINN7-KONS TANK  MANGLER
LD P_On
AND K1_TR06_TID_S  ; KURS 1 TRINN 06 TID
ANDNOT K1_TR07_TID_S  ; KURS 1 TRINN 07TID
OUT TR0
AND T82_KONDLAV_KURSKONTR  ; FOR LAV KONSENTRASJON PAA TANK TIL AA STARTE LUTFASE.
ANDNOT K1_1_VMF_FERDIG
OUT VST80_K1_T82_LAVCOND  ; KURS1  FASE LUT INN KONSENTRASJON T82 FOR LAV
LD TR0
AND T84_KONDLAV_KURSKONTR  ; FOR LAV KONSENTRASJON PAA TANK TIL AA STARTE LUTFASE.
AND K1_1_VMF_FERDIG
OUT VST80_K1_T84_LAVCOND  ; KURS1  FASE LUT INN KONSENTRASJON T84 FOR LAV

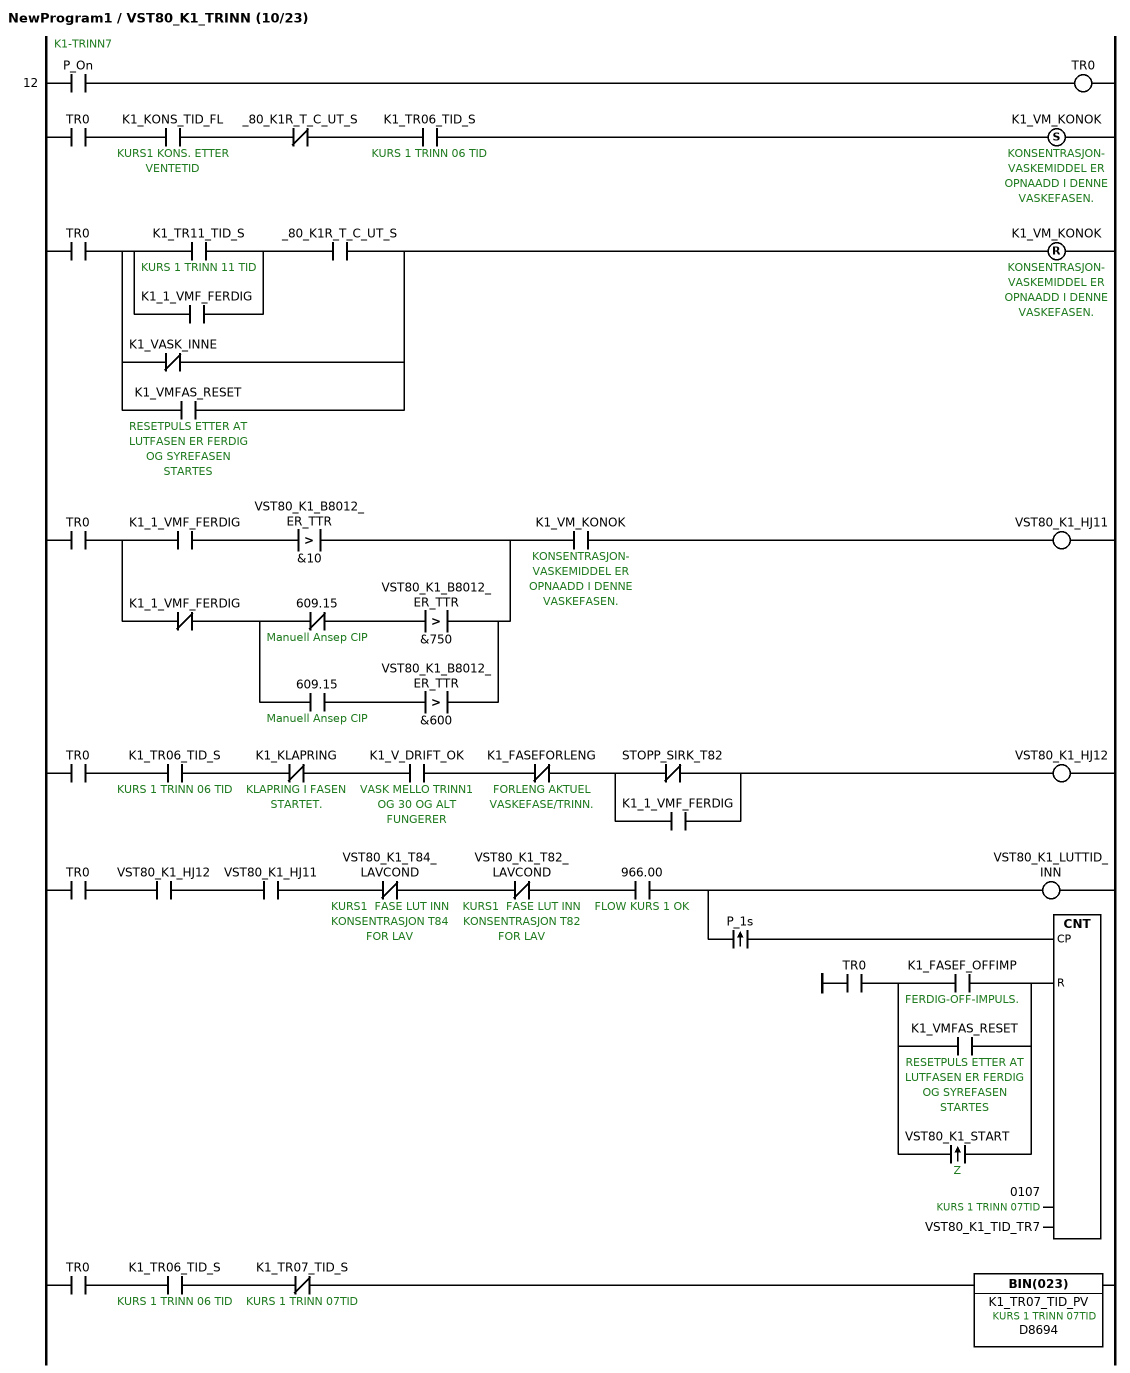
; rung 12: K1-TRINN7
LD P_On
OUT TR0
AND K1_KONS_TID_FL  ; KURS1 KONS. ETTER VENTETID
ANDNOT _80_K1R_T_C_UT_S
AND K1_TR06_TID_S  ; KURS 1 TRINN 06 TID
SET K1_VM_KONOK  ; KONSENTRASJON-VASKEMIDDEL ER OPNAADD I DENNE VASKEFASEN.
LD TR0
LD K1_TR11_TID_S  ; KURS 1 TRINN 11 TID
OR K1_1_VMF_FERDIG
AND _80_K1R_T_C_UT_S
ORNOT K1_VASK_INNE
OR K1_VMFAS_RESET  ; RESETPULS ETTER AT LUTFASEN ER FERDIG OG SYREFASEN STARTES
ANDLD
RSET K1_VM_KONOK  ; KONSENTRASJON-VASKEMIDDEL ER OPNAADD I DENNE VASKEFASEN.
LD TR0
LD K1_1_VMF_FERDIG
AND>(320) VST80_K1_B8012_ER_TTR &10
LDNOT K1_1_VMF_FERDIG
LDNOT 609.15  ; Manuell Ansep CIP
AND>(320) VST80_K1_B8012_ER_TTR &750
LD 609.15  ; Manuell Ansep CIP
AND>(320) VST80_K1_B8012_ER_TTR &600
ORLD
ANDLD
ORLD
ANDLD
AND K1_VM_KONOK  ; KONSENTRASJON-VASKEMIDDEL ER OPNAADD I DENNE VASKEFASEN.
OUT VST80_K1_HJ11
LD TR0
AND K1_TR06_TID_S  ; KURS 1 TRINN 06 TID
ANDNOT K1_KLAPRING  ; KLAPRING I FASEN STARTET.
AND K1_V_DRIFT_OK  ; VASK MELLO TRINN1 OG 30 OG ALT FUNGERER
ANDNOT K1_FASEFORLENG  ; FORLENG AKTUEL VASKEFASE/TRINN.
LDNOT STOPP_SIRK_T82
OR K1_1_VMF_FERDIG
ANDLD
OUT VST80_K1_HJ12
LD TR0
AND VST80_K1_HJ12
AND VST80_K1_HJ11
ANDNOT VST80_K1_T84_LAVCOND  ; KURS1  FASE LUT INN KONSENTRASJON T84 FOR LAV
ANDNOT VST80_K1_T82_LAVCOND  ; KURS1  FASE LUT INN KONSENTRASJON T82 FOR LAV
AND 966.00  ; FLOW KURS 1 OK
OUT VST80_K1_LUTTID_INN
@AND P_1s
LD TR0
LD K1_FASEF_OFFIMP  ; FERDIG-OFF-IMPULS.
OR K1_VMFAS_RESET  ; RESETPULS ETTER AT LUTFASEN ER FERDIG OG SYREFASEN STARTES
@OR VST80_K1_START  ; Z
ANDLD
CNT 0107 VST80_K1_TID_TR7  ; KURS 1 TRINN 07TID
LD TR0
AND K1_TR06_TID_S  ; KURS 1 TRINN 06 TID
ANDNOT K1_TR07_TID_S  ; KURS 1 TRINN 07TID
BIN(023) K1_TR07_TID_PV D8694  ; KURS 1 TRINN 07TID

